// TIA Portal V20 export
VAR_GLOBAL   // PLC tag table "Kraft"
   Temperature_Read AT %IW1000 : Int;
   Temperature_Set AT %IW1002 : Int;
   Humidity_Read AT %IW1004 : Int;
END_VAR
